PROGRAM FilterPressureCtrl
VAR
END_VAR

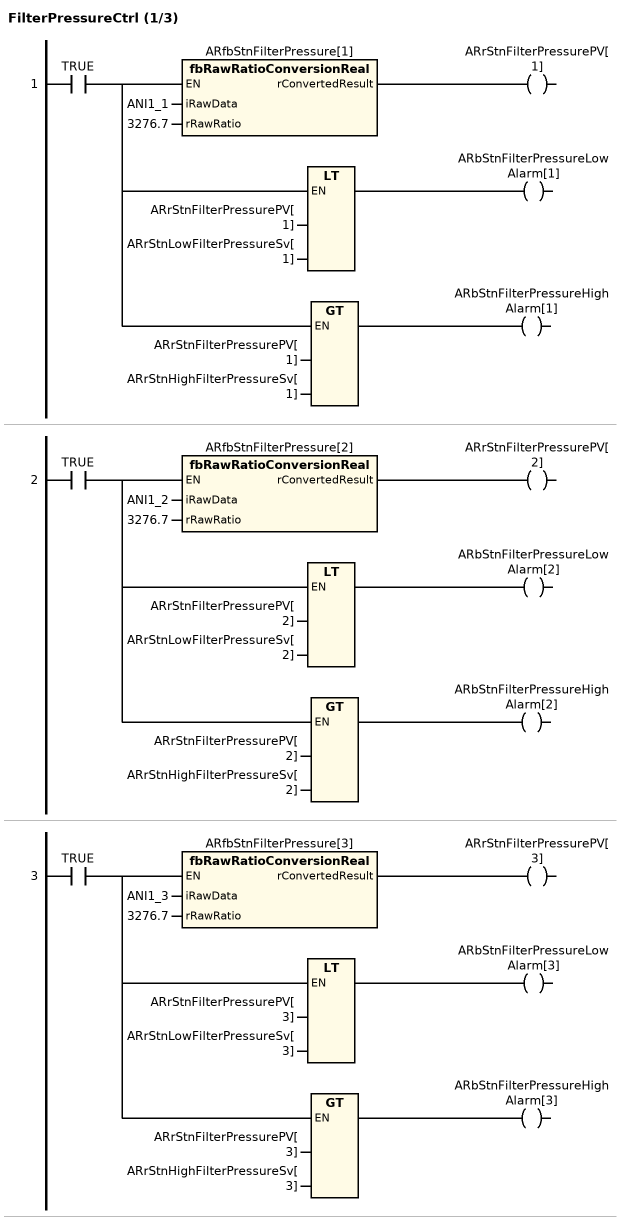
// NETWORK 1
ARfbStnFilterPressure[1](iRawData := ANI1_1, rRawRatio := 3276.7); // fbRawRatioConversionReal
ARrStnFilterPressurePV[1] := ARfbStnFilterPressure[1].rConvertedResult;
ARbStnFilterPressureLowAlarm[1] := ARrStnFilterPressurePV[1] < ARrStnLowFilterPressureSv[1];
ARbStnFilterPressureHighAlarm[1] := ARrStnFilterPressurePV[1] > ARrStnHighFilterPressureSv[1];

// NETWORK 2
ARfbStnFilterPressure[2](iRawData := ANI1_2, rRawRatio := 3276.7); // fbRawRatioConversionReal
ARrStnFilterPressurePV[2] := ARfbStnFilterPressure[2].rConvertedResult;
ARbStnFilterPressureLowAlarm[2] := ARrStnFilterPressurePV[2] < ARrStnLowFilterPressureSv[2];
ARbStnFilterPressureHighAlarm[2] := ARrStnFilterPressurePV[2] > ARrStnHighFilterPressureSv[2];

// NETWORK 3
ARfbStnFilterPressure[3](iRawData := ANI1_3, rRawRatio := 3276.7); // fbRawRatioConversionReal
ARrStnFilterPressurePV[3] := ARfbStnFilterPressure[3].rConvertedResult;
ARbStnFilterPressureLowAlarm[3] := ARrStnFilterPressurePV[3] < ARrStnLowFilterPressureSv[3];
ARbStnFilterPressureHighAlarm[3] := ARrStnFilterPressurePV[3] > ARrStnHighFilterPressureSv[3];

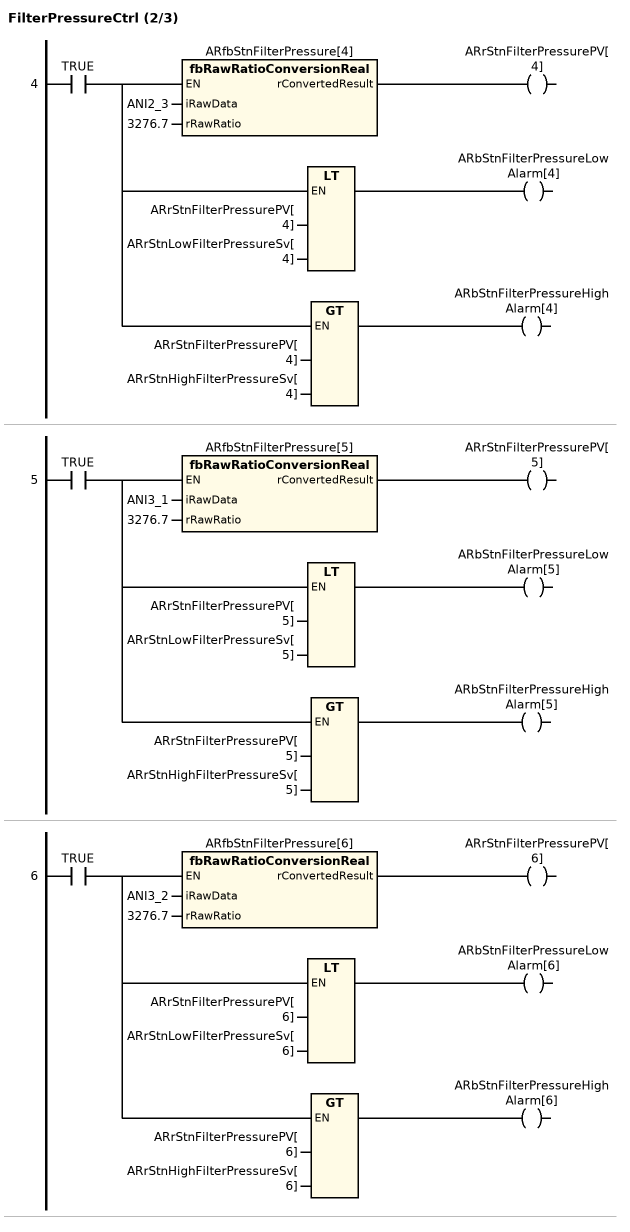
// NETWORK 4
ARfbStnFilterPressure[4](iRawData := ANI2_3, rRawRatio := 3276.7); // fbRawRatioConversionReal
ARrStnFilterPressurePV[4] := ARfbStnFilterPressure[4].rConvertedResult;
ARbStnFilterPressureLowAlarm[4] := ARrStnFilterPressurePV[4] < ARrStnLowFilterPressureSv[4];
ARbStnFilterPressureHighAlarm[4] := ARrStnFilterPressurePV[4] > ARrStnHighFilterPressureSv[4];

// NETWORK 5
ARfbStnFilterPressure[5](iRawData := ANI3_1, rRawRatio := 3276.7); // fbRawRatioConversionReal
ARrStnFilterPressurePV[5] := ARfbStnFilterPressure[5].rConvertedResult;
ARbStnFilterPressureLowAlarm[5] := ARrStnFilterPressurePV[5] < ARrStnLowFilterPressureSv[5];
ARbStnFilterPressureHighAlarm[5] := ARrStnFilterPressurePV[5] > ARrStnHighFilterPressureSv[5];

// NETWORK 6
ARfbStnFilterPressure[6](iRawData := ANI3_2, rRawRatio := 3276.7); // fbRawRatioConversionReal
ARrStnFilterPressurePV[6] := ARfbStnFilterPressure[6].rConvertedResult;
ARbStnFilterPressureLowAlarm[6] := ARrStnFilterPressurePV[6] < ARrStnLowFilterPressureSv[6];
ARbStnFilterPressureHighAlarm[6] := ARrStnFilterPressurePV[6] > ARrStnHighFilterPressureSv[6];

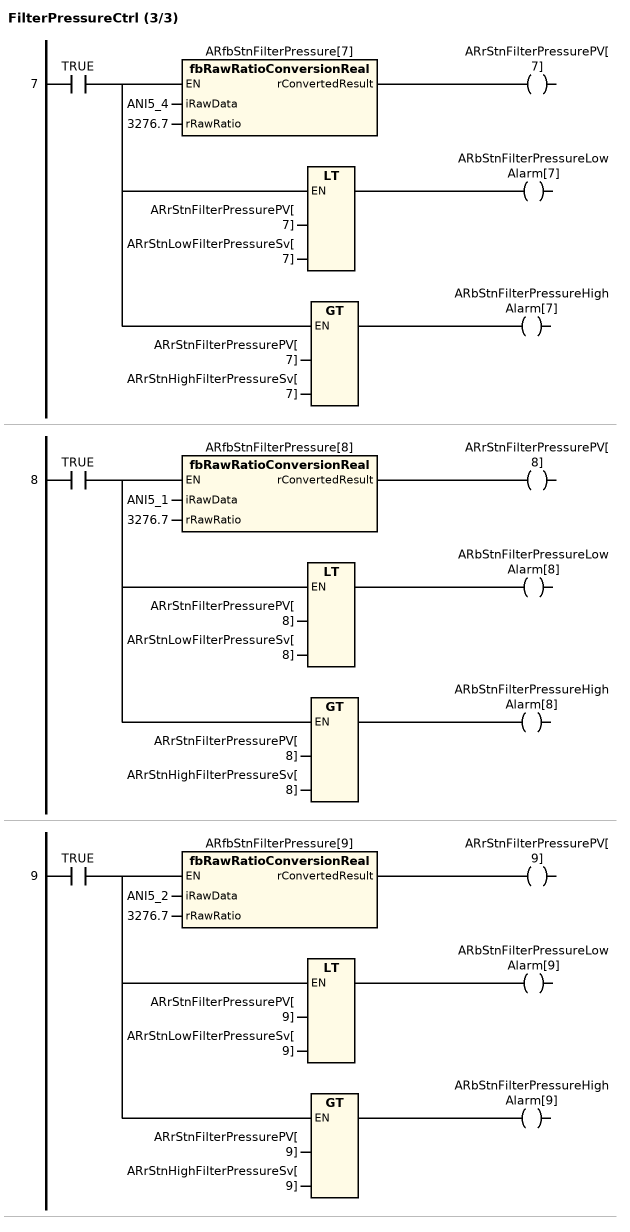
// NETWORK 7
ARfbStnFilterPressure[7](iRawData := ANI5_4, rRawRatio := 3276.7); // fbRawRatioConversionReal
ARrStnFilterPressurePV[7] := ARfbStnFilterPressure[7].rConvertedResult;
ARbStnFilterPressureLowAlarm[7] := ARrStnFilterPressurePV[7] < ARrStnLowFilterPressureSv[7];
ARbStnFilterPressureHighAlarm[7] := ARrStnFilterPressurePV[7] > ARrStnHighFilterPressureSv[7];

// NETWORK 8
ARfbStnFilterPressure[8](iRawData := ANI5_1, rRawRatio := 3276.7); // fbRawRatioConversionReal
ARrStnFilterPressurePV[8] := ARfbStnFilterPressure[8].rConvertedResult;
ARbStnFilterPressureLowAlarm[8] := ARrStnFilterPressurePV[8] < ARrStnLowFilterPressureSv[8];
ARbStnFilterPressureHighAlarm[8] := ARrStnFilterPressurePV[8] > ARrStnHighFilterPressureSv[8];

// NETWORK 9
ARfbStnFilterPressure[9](iRawData := ANI5_2, rRawRatio := 3276.7); // fbRawRatioConversionReal
ARrStnFilterPressurePV[9] := ARfbStnFilterPressure[9].rConvertedResult;
ARbStnFilterPressureLowAlarm[9] := ARrStnFilterPressurePV[9] < ARrStnLowFilterPressureSv[9];
ARbStnFilterPressureHighAlarm[9] := ARrStnFilterPressurePV[9] > ARrStnHighFilterPressureSv[9];

END_PROGRAM

(* stored: Version 1.1.0.1, ProductVersion 3.1.4024.12
   POU FilterPressureCtrl: Id {269e1384-60f8-40ae-aa3c-cd75fb1368dd}, SpecialFunc None *)
